PROGRAM PRG_PLAS_19_CompleteOuterCtrl
VAR
	rsCompleteOCVData				: RS;
	fbCompleteOCV  					: FB_T04_CompleteOCV;

	fbDebugCNT				: FB_DEBUG_CounterArray;
	aCNTDebug				: ARRAY [1..10] OF UDINT;
	bResetCNT					: BOOL;

	ctuConsecutiveIntermediateNoRead		: CTU;
	ctuConsecutiveOCVMissing		: CTU;
END_VAR

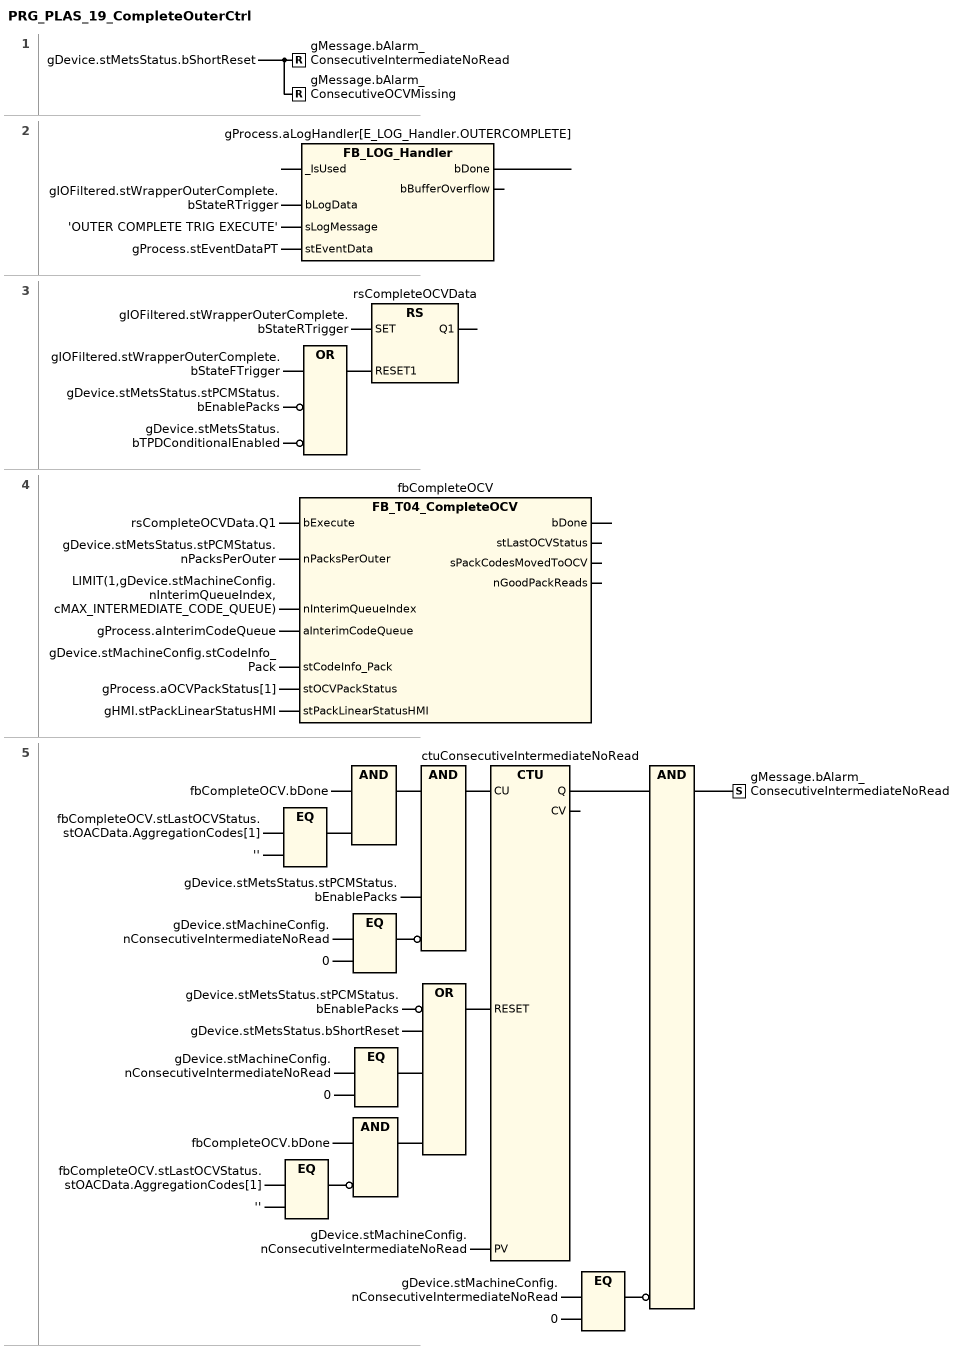
// NETWORK 1
gMessage.bAlarm_ConsecutiveIntermediateNoRead R= gDevice.stMetsStatus.bShortReset;
gMessage.bAlarm_ConsecutiveOCVMissing R= gDevice.stMetsStatus.bShortReset;

// NETWORK 2
gProcess.aLogHandler[E_LOG_Handler.OUTERCOMPLETE](
    bLogData := gIOFiltered.stWrapperOuterComplete.bStateRTrigger,
    sLogMessage := 'OUTER COMPLETE TRIG EXECUTE',
    stEventData := gProcess.stEventDataPT); // FB_LOG_Handler

// NETWORK 3
rsCompleteOCVData(SET := gIOFiltered.stWrapperOuterComplete.bStateRTrigger, RESET1 := gIOFiltered.stWrapperOuterComplete.bStateFTrigger OR NOT gDevice.stMetsStatus.stPCMStatus.bEnablePacks OR NOT gDevice.stMetsStatus.bTPDConditionalEnabled); // RS

// NETWORK 4
fbCompleteOCV(
    bExecute := rsCompleteOCVData.Q1,
    nPacksPerOuter := gDevice.stMetsStatus.stPCMStatus.nPacksPerOuter,
    nInterimQueueIndex := LIMIT(1,gDevice.stMachineConfig.nInterimQueueIndex, cMAX_INTERMEDIATE_CODE_QUEUE),
    aInterimCodeQueue := gProcess.aInterimCodeQueue,
    stCodeInfo_Pack := gDevice.stMachineConfig.stCodeInfo_Pack,
    stOCVPackStatus := gProcess.aOCVPackStatus[1],
    stPackLinearStatusHMI := gHMI.stPackLinearStatusHMI); // FB_T04_CompleteOCV

// NETWORK 5
ctuConsecutiveIntermediateNoRead(
    CU := (fbCompleteOCV.bDone AND fbCompleteOCV.stLastOCVStatus.stOACData.AggregationCodes[1] = '') AND gDevice.stMetsStatus.stPCMStatus.bEnablePacks AND NOT (gDevice.stMachineConfig.nConsecutiveIntermediateNoRead = 0),
    RESET := NOT gDevice.stMetsStatus.stPCMStatus.bEnablePacks OR gDevice.stMetsStatus.bShortReset OR gDevice.stMachineConfig.nConsecutiveIntermediateNoRead = 0 OR fbCompleteOCV.bDone AND NOT (fbCompleteOCV.stLastOCVStatus.stOACData.AggregationCodes[1] = ''),
    PV := gDevice.stMachineConfig.nConsecutiveIntermediateNoRead); // CTU
gMessage.bAlarm_ConsecutiveIntermediateNoRead S= ctuConsecutiveIntermediateNoRead.Q AND NOT (gDevice.stMachineConfig.nConsecutiveIntermediateNoRead = 0);

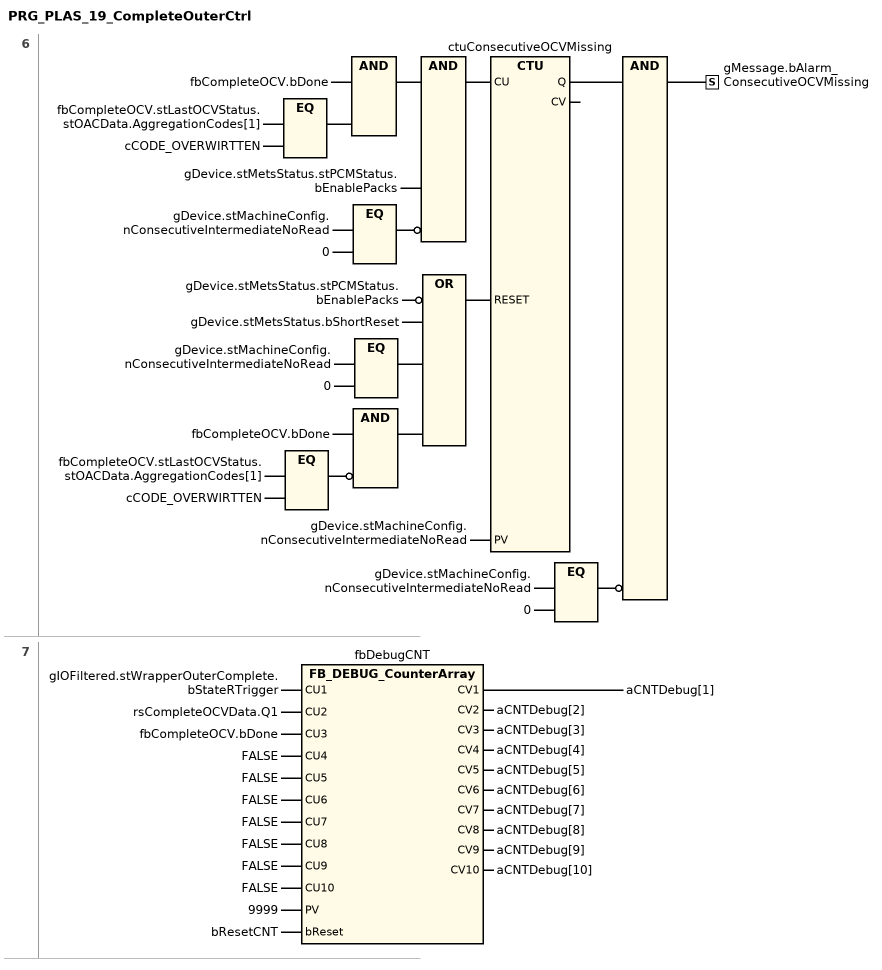
// NETWORK 6
ctuConsecutiveOCVMissing(
    CU := (fbCompleteOCV.bDone AND fbCompleteOCV.stLastOCVStatus.stOACData.AggregationCodes[1] = cCODE_OVERWIRTTEN) AND gDevice.stMetsStatus.stPCMStatus.bEnablePacks AND NOT (gDevice.stMachineConfig.nConsecutiveIntermediateNoRead = 0),
    RESET := NOT gDevice.stMetsStatus.stPCMStatus.bEnablePacks OR gDevice.stMetsStatus.bShortReset OR gDevice.stMachineConfig.nConsecutiveIntermediateNoRead = 0 OR fbCompleteOCV.bDone AND NOT (fbCompleteOCV.stLastOCVStatus.stOACData.AggregationCodes[1] = cCODE_OVERWIRTTEN),
    PV := gDevice.stMachineConfig.nConsecutiveIntermediateNoRead); // CTU
gMessage.bAlarm_ConsecutiveOCVMissing S= ctuConsecutiveOCVMissing.Q AND NOT (gDevice.stMachineConfig.nConsecutiveIntermediateNoRead = 0);

// NETWORK 7
fbDebugCNT(
    CU1 := gIOFiltered.stWrapperOuterComplete.bStateRTrigger,
    CU2 := rsCompleteOCVData.Q1,
    CU3 := fbCompleteOCV.bDone,
    CU4 := FALSE,
    CU5 := FALSE,
    CU6 := FALSE,
    CU7 := FALSE,
    CU8 := FALSE,
    CU9 := FALSE,
    CU10 := FALSE,
    PV := 9999,
    bReset := bResetCNT,
    CV2 => aCNTDebug[2],
    CV3 => aCNTDebug[3],
    CV4 => aCNTDebug[4],
    CV5 => aCNTDebug[5],
    CV6 => aCNTDebug[6],
    CV7 => aCNTDebug[7],
    CV8 => aCNTDebug[8],
    CV9 => aCNTDebug[9],
    CV10 => aCNTDebug[10]); // FB_DEBUG_CounterArray
aCNTDebug[1] := fbDebugCNT.CV1;

END_PROGRAM

(* stored: Version 1.1.0.1
   POU PRG_PLAS_19_CompleteOuterCtrl: Id {de24b5c6-2b87-4d30-a2f2-efe53e0bbf69}, SpecialFunc None *)
